// TIA Portal V20 export
ORGANIZATION_BLOCK "MC_PreServo"   // OB67, LAD, PreServo
// stored: SetENOAutomatically false
   VAR_INPUT
      Initial_Call : Bool;
      PIP_Input : Bool;
      PIP_Output : Bool;
      IO_System : USInt;
      Event_Count : Int;
      Synchronous : Bool;
      CycleTime : UDInt;
   END_VAR
BEGIN

REGION Network 1: Simulation
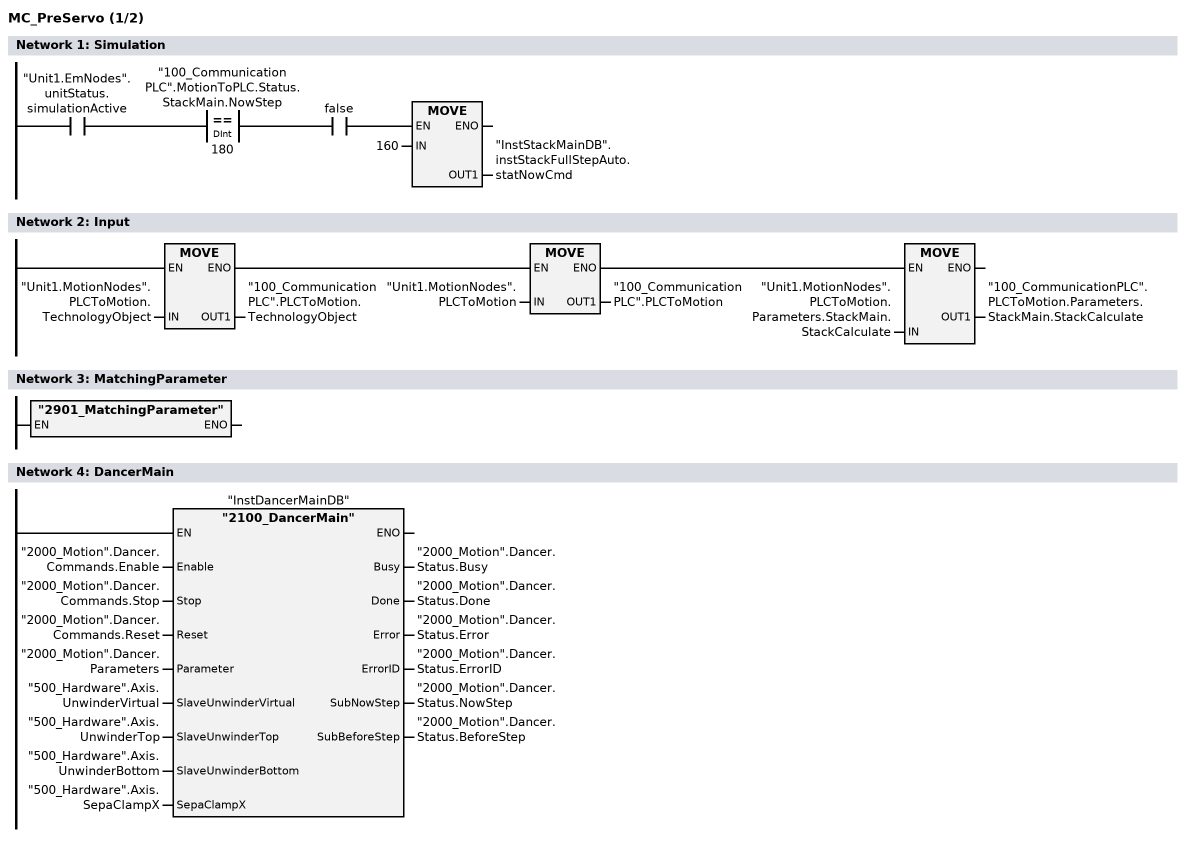
   RUNG wire#powerrail
      Contact( "Unit1.EmNodes".unitStatus.simulationActive )
      { S7_Templates := "SrcType := DInt" } EQ_Contact(in1 := "100_CommunicationPLC".MotionToPLC.Status.StackMain.NowStep, in2 := 180)
      Contact( false )
      Move(in := 160, out1 => "InstStackMainDB".instStackFullStepAuto.statNowCmd)
   END_RUNG
   // the same network as SCL:
   IF "Unit1.EmNodes".unitStatus.simulationActive AND ("100_CommunicationPLC".MotionToPLC.Status.StackMain.NowStep = 180) AND false THEN
       "InstStackMainDB".instStackFullStepAuto.statNowCmd := 160;
   END_IF;
END_REGION

REGION Network 2: Input
   RUNG wire#powerrail
      Move(in := "Unit1.MotionNodes".PLCToMotion.TechnologyObject, out1 => "100_CommunicationPLC".PLCToMotion.TechnologyObject)
      Move(in := "Unit1.MotionNodes".PLCToMotion, out1 => "100_CommunicationPLC".PLCToMotion)
      Move(in := "Unit1.MotionNodes".PLCToMotion.Parameters.StackMain.StackCalculate, out1 => "100_CommunicationPLC".PLCToMotion.Parameters.StackMain.StackCalculate)
   END_RUNG
   // the same network as SCL:
   "100_CommunicationPLC".PLCToMotion.TechnologyObject := "Unit1.MotionNodes".PLCToMotion.TechnologyObject;
   "100_CommunicationPLC".PLCToMotion := "Unit1.MotionNodes".PLCToMotion;
   "100_CommunicationPLC".PLCToMotion.Parameters.StackMain.StackCalculate := "Unit1.MotionNodes".PLCToMotion.Parameters.StackMain.StackCalculate;
END_REGION

REGION Network 3: MatchingParameter
   RUNG wire#powerrail
      "2901_MatchingParameter"()
   END_RUNG
   // the same network as SCL:
   "2901_MatchingParameter"();
END_REGION

REGION Network 4: DancerMain
   RUNG wire#powerrail
      "InstDancerMainDB"(Enable := "2000_Motion".Dancer.Commands.Enable, Stop := "2000_Motion".Dancer.Commands.Stop, Reset := "2000_Motion".Dancer.Commands.Reset, Parameter := "2000_Motion".Dancer.Parameters, SlaveUnwinderVirtual := "500_Hardware".Axis.UnwinderVirtual, SlaveUnwinderTop := "500_Hardware".Axis.UnwinderTop, SlaveUnwinderBottom := "500_Hardware".Axis.UnwinderBottom, SepaClampX := "500_Hardware".Axis.SepaClampX, Busy => "2000_Motion".Dancer.Status.Busy, Done => "2000_Motion".Dancer.Status.Done, Error => "2000_Motion".Dancer.Status.Error, ErrorID => "2000_Motion".Dancer.Status.ErrorID, SubNowStep => "2000_Motion".Dancer.Status.NowStep, SubBeforeStep => "2000_Motion".Dancer.Status.BeforeStep)
   END_RUNG
   // the same network as SCL:
   "InstDancerMainDB"(Enable := "2000_Motion".Dancer.Commands.Enable,   // "2100_DancerMain"
                      Stop := "2000_Motion".Dancer.Commands.Stop,
                      Reset := "2000_Motion".Dancer.Commands.Reset,
                      Parameter := "2000_Motion".Dancer.Parameters,
                      SlaveUnwinderVirtual := "500_Hardware".Axis.UnwinderVirtual,
                      SlaveUnwinderTop := "500_Hardware".Axis.UnwinderTop,
                      SlaveUnwinderBottom := "500_Hardware".Axis.UnwinderBottom,
                      SepaClampX := "500_Hardware".Axis.SepaClampX,
                      Busy => "2000_Motion".Dancer.Status.Busy,
                      Done => "2000_Motion".Dancer.Status.Done,
                      Error => "2000_Motion".Dancer.Status.Error,
                      ErrorID => "2000_Motion".Dancer.Status.ErrorID,
                      SubNowStep => "2000_Motion".Dancer.Status.NowStep,
                      SubBeforeStep => "2000_Motion".Dancer.Status.BeforeStep);
END_REGION

REGION Network 5: StackMain
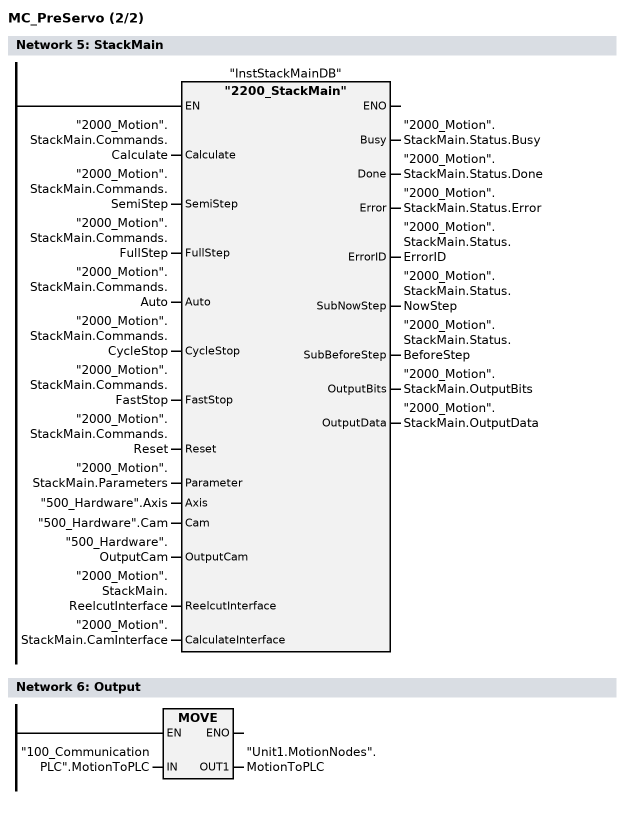
   RUNG wire#powerrail
      "InstStackMainDB"(Calculate := "2000_Motion".StackMain.Commands.Calculate, SemiStep := "2000_Motion".StackMain.Commands.SemiStep, FullStep := "2000_Motion".StackMain.Commands.FullStep, Auto := "2000_Motion".StackMain.Commands.Auto, CycleStop := "2000_Motion".StackMain.Commands.CycleStop, FastStop := "2000_Motion".StackMain.Commands.FastStop, Reset := "2000_Motion".StackMain.Commands.Reset, Parameter := "2000_Motion".StackMain.Parameters, Axis := "500_Hardware".Axis, Cam := "500_Hardware".Cam, OutputCam := "500_Hardware".OutputCam, ReelcutInterface := "2000_Motion".StackMain.ReelcutInterface, CalculateInterface := "2000_Motion".StackMain.CamInterface, Busy => "2000_Motion".StackMain.Status.Busy, Done => "2000_Motion".StackMain.Status.Done, Error => "2000_Motion".StackMain.Status.Error, ErrorID => "2000_Motion".StackMain.Status.ErrorID, SubNowStep => "2000_Motion".StackMain.Status.NowStep, SubBeforeStep => "2000_Motion".StackMain.Status.BeforeStep, OutputBits => "2000_Motion".StackMain.OutputBits, OutputData => "2000_Motion".StackMain.OutputData)
   END_RUNG
   // the same network as SCL:
   "InstStackMainDB"(Calculate := "2000_Motion".StackMain.Commands.Calculate,   // "2200_StackMain"
                     SemiStep := "2000_Motion".StackMain.Commands.SemiStep,
                     FullStep := "2000_Motion".StackMain.Commands.FullStep,
                     Auto := "2000_Motion".StackMain.Commands.Auto,
                     CycleStop := "2000_Motion".StackMain.Commands.CycleStop,
                     FastStop := "2000_Motion".StackMain.Commands.FastStop,
                     Reset := "2000_Motion".StackMain.Commands.Reset,
                     Parameter := "2000_Motion".StackMain.Parameters,
                     Axis := "500_Hardware".Axis,
                     Cam := "500_Hardware".Cam,
                     OutputCam := "500_Hardware".OutputCam,
                     ReelcutInterface := "2000_Motion".StackMain.ReelcutInterface,
                     CalculateInterface := "2000_Motion".StackMain.CamInterface,
                     Busy => "2000_Motion".StackMain.Status.Busy,
                     Done => "2000_Motion".StackMain.Status.Done,
                     Error => "2000_Motion".StackMain.Status.Error,
                     ErrorID => "2000_Motion".StackMain.Status.ErrorID,
                     SubNowStep => "2000_Motion".StackMain.Status.NowStep,
                     SubBeforeStep => "2000_Motion".StackMain.Status.BeforeStep,
                     OutputBits => "2000_Motion".StackMain.OutputBits,
                     OutputData => "2000_Motion".StackMain.OutputData);
END_REGION

REGION Network 6: Output
   RUNG wire#powerrail
      Move(in := "100_CommunicationPLC".MotionToPLC, out1 => "Unit1.MotionNodes".MotionToPLC)
   END_RUNG
   // the same network as SCL:
   "Unit1.MotionNodes".MotionToPLC := "100_CommunicationPLC".MotionToPLC;
END_REGION
END_ORGANIZATION_BLOCK
